(* CODESYS project Admin.xml

Project tree, tasks and I/O mapping:
  program Admin [LD]
*)

// Admin
PROGRAM Admin
VAR_INPUT
	LoadDefaults: BOOL;
END_VAR
VAR
	_ResetBaggerSettings: BOOL;
END_VAR
VAR // added by the converter: edge detectors and wires of the graphical bodies
    _rt1, _rt2 : R_TRIG;
END_VAR

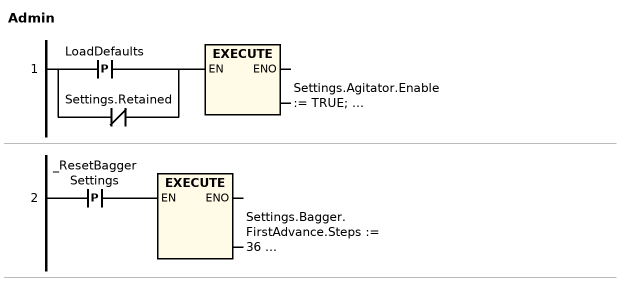
// NETWORK 1
_rt1(CLK := LoadDefaults);
IF _rt1.Q OR NOT Settings.Retained THEN
    Settings.Agitator.Enable := TRUE;
    Settings.Agitator.AutoAgitate := TRUE;
    Settings.Agitator.ReverseTime := T#10S;
    Settings.Agitator.DwellTime := T#3S;
    Settings.Agitator.ForwardTime := T#2S;
    Settings.Agitator.IdleTime := T#15M;
    
    Settings.Bagger.FirstAdvance.Steps := 3600;
    Settings.Bagger.FirstAdvance.Direction := 1;
    Settings.Bagger.FirstAdvance.Speed := 500;
    Settings.Bagger.FirstRetract.Steps := 600;
    Settings.Bagger.FirstRetract.Direction := 0;
    Settings.Bagger.FirstRetract.Speed := 500;
    Settings.Bagger.RetryAdvance.Steps := 600;
    Settings.Bagger.RetryAdvance.Direction := 1;
    Settings.Bagger.RetryAdvance.Speed := 500;
    Settings.Bagger.RetryRetract.Steps := 600;
    Settings.Bagger.RetryRetract.Direction := 0;
    Settings.Bagger.RetryRetract.Speed := 500;
    Settings.Bagger.TearRetract.Steps := 300;
    Settings.Bagger.TearRetract.Direction := 0;
    Settings.Bagger.TearRetract.Speed := 300;
    Settings.Bagger.ResetBag.Steps := 1000;
    Settings.Bagger.ResetBag.Direction := 1;
    Settings.Bagger.ResetBag.Speed := 100;
    Settings.Bagger.RetractOneBag.Steps := 3200;
    Settings.Bagger.RetractOneBag.Direction := 0;
    Settings.Bagger.RetractOneBag.Speed := 300;
    Settings.Bagger.MaxBagOpenRetries := 5;
    Settings.Bagger.MaxBagRetries := 3;
    
    Settings.Door.ManualUnlock := FALSE;
    Settings.Door.AutoDoorLock := TRUE;
    Settings.Door.IgnoreKicker := FALSE;
    Settings.Door.CheckLockDelay := T#1S;
    
    Settings.Heater.Enable := TRUE;
    Settings.Heater.MinTemp := 70.0;
    Settings.Heater.LowPoint := 75.0;
    Settings.Heater.SetPoint := 80.0;
    Settings.Heater.MaxTemp := 100.0;
    Settings.Heater.Timeout := T#3M;
    Settings.Heater.ResetTimeout := FALSE;
    
    Settings.HeatSeal.Enable := TRUE;
    Settings.HeatSeal.SealingTime := T#3S;
    
    Settings.Hopper.Enable := TRUE;
    
    Settings.IceFeed.Enable := TRUE;
    Settings.IceFeed.MaxFeedTime := T#10S;
    Settings.IceFeed.TopOffTime := T#2S;
    
    Settings.IceMaker.Enable := TRUE;
    Settings.IceMaker.MakeIceTimeout := T#2H;
    
    Settings.Kicker.Enable := TRUE;
    
    // Motors
    Settings.AgitatorMotor.Override := FALSE;
    Settings.AgitatorMotor.OverrideMotor := FALSE;
    Settings.AgitatorMotor.OverrideReverse := FALSE;
    Settings.AgitatorMotor.Speed := 50;
    
    Settings.BagFeedMotor.Enable := TRUE;
    Settings.BagFeedMotor.InputFunction := 1;
    Settings.BagFeedMotor.CounterLimit := 30;
    Settings.BagFeedMotor.RateTime := 1000;
    Settings.BagFeedMotor.RateChannel := 1;
    Settings.BagFeedMotor.Speed := 50;
    //Settings.BagFeedMotor.GearRatio := 200;
    //Settings.BagFeedMotor.PPR := 30;
    Settings.BagFeedMotor.MaxRPM := 4000;
    Settings.BagFeedMotor.CounterCommand := 0;
    Settings.BagFeedMotor.KP := 12;
    Settings.BagFeedMotor.TN := 1;
    Settings.BagFeedMotor.TV := 0;
    Settings.BagFeedMotor.Y_MIN := 30;
    Settings.BagFeedMotor.Y_MAX := 1000;
    //Settings.BagFeedMotor.BagLengthPulses := 3000;
    
    Settings.BlowerMotor.Override := FALSE;
    Settings.BlowerMotor.OverrideMotor := FALSE;
    
    Settings.HeatSealMotor.Override := FALSE;
    Settings.HeatSealMotor.OverrideMotor := FALSE;
    Settings.HeatSealMotor.OverrideReverse := FALSE;
    Settings.HeatSealMotor.OverrideBrake := FALSE;
    
    Settings.IceFeedMotor.Override := FALSE;
    Settings.IceFeedMotor.OverrideMotor := FALSE;
    
    Settings.KickerMotor.Override := FALSE;
    Settings.KickerMotor.OverrideMotor := FALSE;
    Settings.KickerMotor.OverrideBrake := FALSE;
    
    // Sensors
    Settings.BagFullSensor.OffDelay := T#0MS;
    Settings.BagFullSensor.OnDelay := T#0MS;
    
    Settings.BagLabelSensor.OffDelay := T#0MS;
    Settings.BagLabelSensor.OnDelay := T#0MS;
    
    Settings.BagOpenSensor.OffDelay := T#0MS;
    Settings.BagOpenSensor.OnDelay := T#0MS;
    
    Settings.DoorClosedSensor.OffDelay := T#0MS;
    Settings.DoorClosedSensor.OnDelay := T#250MS;
    
    Settings.DoorLockedSensor.OffDelay := T#0MS;
    Settings.DoorLockedSensor.OnDelay := T#0MS;
    
    Settings.HeatSealClosedSensor.OffDelay := T#0MS;
    Settings.HeatSealClosedSensor.OnDelay := T#0MS;
    
    Settings.HeatSealOpenSensor.OffDelay := T#0MS;
    Settings.HeatSealOpenSensor.OnDelay := T#0MS;
    
    Settings.HopperMaximumSensor.OffDelay := T#1000MS;
    Settings.HopperMaximumSensor.OnDelay := T#500MS;
    
    Settings.HopperMinimumSensor.OffDelay := T#1000MS;
    Settings.HopperMinimumSensor.OnDelay := T#500MS;
    
    Settings.KickerBlockedSensor.OffDelay := T#1000MS;
    Settings.KickerBlockedSensor.OnDelay := T#0MS;
    
    Settings.KickerDownSensor.OffDelay := T#0MS;
    Settings.KickerDownSensor.OnDelay := T#0MS;
    
    Settings.KickerUpSensor.OffDelay := T#0MS;
    Settings.KickerUpSensor.OnDelay := T#0MS;
    
    Settings.Retained := TRUE;
END_IF

// NETWORK 2
_rt2(CLK := _ResetBaggerSettings);
IF _rt2.Q THEN
    Settings.Bagger.FirstAdvance.Steps := 3600;
    Settings.Bagger.FirstAdvance.Direction := 1;
    Settings.Bagger.FirstAdvance.Speed := 500;
    Settings.Bagger.FirstRetract.Steps := 600;
    Settings.Bagger.FirstRetract.Direction := 0;
    Settings.Bagger.FirstRetract.Speed := 500;
    Settings.Bagger.RetryAdvance.Steps := 600;
    Settings.Bagger.RetryAdvance.Direction := 1;
    Settings.Bagger.RetryAdvance.Speed := 500;
    Settings.Bagger.RetryRetract.Steps := 600;
    Settings.Bagger.RetryRetract.Direction := 0;
    Settings.Bagger.RetryRetract.Speed := 500;
    Settings.Bagger.TearRetract.Steps := 300;
    Settings.Bagger.TearRetract.Direction := 0;
    Settings.Bagger.TearRetract.Speed := 300;
    Settings.Bagger.ResetBag.Steps := 1000;
    Settings.Bagger.ResetBag.Direction := 1;
    Settings.Bagger.ResetBag.Speed := 100;
    Settings.Bagger.RetractOneBag.Steps := 3200;
    Settings.Bagger.RetractOneBag.Direction := 0;
    Settings.Bagger.RetractOneBag.Speed := 300;
    Settings.Bagger.MaxBagOpenRetries := 5;
    Settings.Bagger.MaxBagRetries := 3;
END_IF

END_PROGRAM
